PROGRAM MAIN
VAR
	
END_VAR

P_Linked_List_Example();

END_PROGRAM

(* stored: Version 1.1.0.1, ProductVersion 3.1.4024.4
   POU MAIN: Id {86dc0999-fc6b-4ce8-a12d-7649401b850c}, SpecialFunc None *)
